// TIA Portal V19 export
FUNCTION "DI WATER TRANSFER" : Void   // FC16, LAD
{ S7_Optimized_Access := 'TRUE' }
// stored: SetENOAutomatically false
BEGIN

REGION Network 1
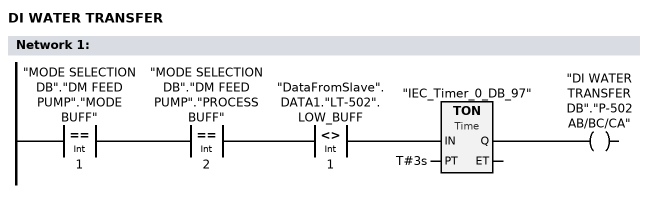
   RUNG wire#powerrail
      { S7_Templates := "SrcType := Int" } EQ_Contact(in1 := "MODE SELECTION DB"."DM FEED PUMP"."MODE BUFF", in2 := 1)
      { S7_Templates := "SrcType := Int" } EQ_Contact(in1 := "MODE SELECTION DB"."DM FEED PUMP"."PROCESS BUFF", in2 := 2)
      { S7_Templates := "SrcType := Int" } NE_Contact(in1 := "DataFromSlave".DATA1."LT-502".LOW_BUFF, in2 := 1)
      { S7_Templates := "time_type := Time" } "IEC_Timer_0_DB_97".TON(pt := T#3s, et =>)
      Coil( "DI WATER TRANSFER DB"."P-502 AB/BC/CA" )
   END_RUNG
   // the same network as SCL:
   "IEC_Timer_0_DB_97".TON(IN := ("MODE SELECTION DB"."DM FEED PUMP"."MODE BUFF" = 1) AND ("MODE SELECTION DB"."DM FEED PUMP"."PROCESS BUFF" = 2) AND ("DataFromSlave".DATA1."LT-502".LOW_BUFF <> 1),
                           PT := T#3s);
   "DI WATER TRANSFER DB"."P-502 AB/BC/CA" := "IEC_Timer_0_DB_97".Q;
END_REGION
END_FUNCTION
